// TIA Portal V17 export
// export: Created 2023-02-25T14:38:25.4831182Z, ExportSetting WithDefaults, DisplayName Totally Integrated Automation Portal, DisplayVersion V17, DisplayName TIA Portal Openness, DisplayVersion V17, DisplayName TIA Portal Version Control Interface, DisplayVersion V17, DisplayName TIA Portal Test Suite Advanced, DisplayVersion V17, DisplayName STEP 7 Professional, DisplayVersion V17, DisplayName SIMATIC Energy Suite, DisplayVersion V17, DisplayName STEP 7 Safety, DisplayVersion V17, DisplayName WinCC Professional, DisplayVersion V17
DATA_BLOCK "HW_MotorControle_DB_1"   // DB8
VERSION : 0.1
// stored: AutoNumber true, InstanceOfName HW_MotorControle, InstanceOfType FB
"HW_MotorControle"
   // VAR_INPUT
   //    inConveyor : "stt_Motor";
   //    FirstScan : Bool;
   // END_VAR
   // VAR_OUTPUT
   //    Conveyor : Real;
   // END_VAR
   // VAR
   //    S1 : Bool;
   //    S2 : Bool;
   //    S3 : Bool;
   //    S4 : Bool;
   //    S5 : Bool;
   //    t1 : Bool;
   //    t2 : Bool;
   //    speedLeft : Real;
   //    IEC_Timer_0_Instance { ExternalAccessible := 'False'; ExternalVisible := 'False'; ExternalWritable := 'False'} : TON_TIME;
   //    IEC_Timer_0_Instance_1 { ExternalAccessible := 'False'; ExternalVisible := 'False'; ExternalWritable := 'False'} : TON_TIME;
   // END_VAR
BEGIN
END_DATA_BLOCK
